TYPE ST_System_MVKW_Parameter :
STRUCT
	AutoQuittierung			: BOOL;
END_STRUCT
END_TYPE

(* stored: Version 1.1.0.1, ProductVersion 3.1.4024.9
   DUT ST_System_MVKW_Parameter: Id {fe972056-0846-4b36-a837-fecf205b837f} *)
